PROGRAM Main
VAR
	// Digital output variables (linked to EL2809 outputs)
	Relay1_Forward : BOOL := FALSE; // Forward relay for Actuator 1
	Relay1_Reverse : BOOL := FALSE; // Reverse relay for Actuator 1
	Relay2_Forward : BOOL := FALSE; // Forward relay for Actuator 2
	Relay2_Reverse : BOOL := FALSE; // Reverse relay for Actuator 2
	
	Actuator1 : FB_LinearActuator;
	bactivation : INT;
	bEnable : BOOL := TRUE;          // General enable for actuators
END_VAR

Actuator1.bRelayForward := ADR(Relay1_Forward);
Actuator1.bRelayReverse := ADR(Relay1_Reverse);

IF bActivation = 1 THEN
// Enable both actuators
Actuator1.Enable(bEnableCmd := bEnable);
END_IF;

IF bActivation = 2 THEN
// Move Actuator 1 forward
Actuator1.MoveForward(bStart := TRUE);
END_IF;

IF bActivation = 3 THEN
// Stop Actuator 1
Actuator1.Stop();
END_IF;

END_PROGRAM

(* stored: Version 1.1.0.1, ProductVersion 3.1.4024.14
   POU MAIN: Id {2bb03cb5-93a9-436f-aabc-0b71ea976dc6}, SpecialFunc None *)
